INTERFACE I_Deserializer

METHOD PUBLIC TryGetBool : BOOL
VAR_INPUT
	Destination : REFERENCE TO BOOL;
END_VAR
END_METHOD

END_INTERFACE

(* stored: Version 1.1.0.1, ProductVersion 3.1.4024.12
   Itf I_Deserializer: Id {9a809a47-2d37-4dd0-9245-adb664c7ec81}
   Method TryGetBool: Id {33323d35-ea95-4530-a59d-9479abb8d2df} *)
